FUNCTION_BLOCK FB_TVRModbusMaster
VAR_INPUT
END_VAR
VAR_OUTPUT
END_VAR
VAR
	fbModbusRTUMaster : ModbusRtuMaster_KL6x22B;	//Modbus RTU Master
	
	nUnitID			:	BYTE :=	0;	//Modbus device ID
	
	//Modbus Registers
	nRegSetpoint	:	WORD := 0;
	nRegForce		:	WORD := 1;
	nRegActual		:	WORD := 7;
	
	//Properties
	bError 			: 	BOOL := FALSE;
	fNominalVolFlow	: 	REAL := 3690;
	fVolFlowSet 	: 	REAL := 0;
	fVolFlowAct		: 	REAL;
	
	//Internal vars
	bFlagForce		:	BOOL := FALSE;
	bModErr 		: 	BOOL;
	ErrID 			: 	MODBUS_ERRORS;
	fRelFlowMax		:	WORD := 10000;
	fRelFlowMin		:	WORD := 1024;
	nForce			:	WORD := 0;
	fSetModbus		:	WORD := fRelFlowMin;
	sVolFlowAct		: 	WORD;
	
	//Timer
	Tim			:	TON;
	
	//State
	nState		:	INT	:= 1;
	
END_VAR

PROPERTY Error : Bool
GET
Error := THIS^.bError;
END_GET
SET
THIS^.bError := Error;
END_SET
END_PROPERTY

PROPERTY NominalVolumeFlow : REAL
GET
NominalVolumeFlow := THIS^.fNominalVolFlow;
END_GET
SET
THIS^.fNominalVolFlow := NominalVolumeFlow;
END_SET
END_PROPERTY

METHOD Run : BOOL
VAR_INPUT
END_VAR

VAR
	END_I: INT;
END_VAR
Tim(PT:=T#100MS,IN:=TRUE);
	IF Tim.Q THEN
		Tim(IN:=FALSE);

		CASE nState OF
			//Force or release force
			1: //Initialize writing force or release
				IF NOT fbModbusRTUMaster.BUSY THEN
					//IF setpoint is 0, force close ELSE release force mode
					IF fVolFlowSet = 0 OR bFlagForce = TRUE THEN
						//Force close
						nForce := 2;
						//Initialize writing process
						fbModbusRTUMaster.WriteSingleRegister(	UnitID		:=	nUnitID,				//Modbus ID of device
																MBAddr		:=	nRegForce,				//Register address,
																Quantity	:=	1,						//Number of registers to be written
																pMemoryAddr	:=	ADR(nForce),			//Pointer to write data
																cbLength	:=	SIZEOF(fVolFlowSet),	//Size of write data
																Timeout		:=	T#5S,					//Time to wait for the slave to respond
																Execute		:=	TRUE
															);
					ELSE
						//Release force close
						nForce := 0;
						//Initialize writing process
						fbModbusRTUMaster.WriteSingleRegister(	UnitID		:=	nUnitID,				//Modbus ID of device
																MBAddr		:=	nRegForce,				//Register address,
																Quantity	:=	1,						//Number of registers to be written
																pMemoryAddr	:=	ADR(nForce),			//Pointer to write data
																cbLength	:=	SIZEOF(fVolFlowSet),	//Size of write data
																Timeout		:=	T#5S,					//Time to wait for the slave to respond
																Execute		:=	TRUE
															);
					END_IF
				END_IF
				nState := 2;
				Run := FALSE;
				
			2:	//Finish writing force or release
				fbModbusRTUMaster.WriteSingleRegister(Execute:=FALSE, Error=>bModErr, ErrorID=>ErrID);
				IF NOT fbModbusRTUMaster.BUSY THEN
					nState := 3;
				END_IF
				Run := FALSE;
				
			3:	//Setpoint writing
				IF NOT fbModbusRTUMaster.BUSY THEN
					//Check operational limits
					IF fVolFlowSet < fRelFlowMin/fRelFlowMax*fNominalVolFlow THEN
						fVolFlowSet := fRelFlowMin/fRelFlowMax*fNominalVolFlow; //Set to minimum allowed volume flow
					ELSIF fVolFlowSet > fNominalVolFlow THEN
						fVolFlowSet := fNominalVolFlow; //Set to maximum allowed volumen flow
					ELSE
						//do nothing
					END_IF
					//Write setpoint
					//fSetModbus := REAL_TO_WORD(fRelFlowMax*(fVolFlowSet-(fRelFlowMin/fRelFlowMax*fNominalVolFlow))/(fNominalVolFlow-fRelFlowMin));
					fSetModbus := REAL_TO_WORD(fRelFlowMax*fVolFlowSet/fNominalVolFlow);
					//Initialize writing process
					fbModbusRTUMaster.WriteSingleRegister(	UnitID		:=	nUnitID,				//Modbus ID of device
															MBAddr		:=	nRegSetpoint,			//Register address
															Quantity	:=	1,						//Number of registers to be written
															pMemoryAddr	:=	ADR(fSetModbus),		//Pointer to write data
															cbLength	:=	SIZEOF(fSetModbus),		//Size of write data
															Timeout		:=	T#5S,					//Time to wait for the slave to respond
															Execute		:=	TRUE
														);
				END_IF
				nState := 4;
				Run := FALSE;

			4: //Finish writing	
				fbModbusRTUMaster.WriteSingleRegister(Execute:=FALSE, Error=>bModErr, ErrorID=>ErrID);
				IF NOT fbModbusRTUMaster.BUSY THEN
					nState := 5;
				END_IF
				Run := FALSE;
					
			5: //Start reading
				IF NOT fbModbusRTUMaster.BUSY THEN
					//Initialize reading process
					fbModbusRTUMaster.ReadRegs(	UnitID		:=	nUnitID,				//Modbus ID of device
												MBAddr		:=	nRegActual,				//Register address
												Quantity	:=	1,						//Number of registers to be read
												pMemoryAddr	:=	ADR(sVolFlowAct),		//Pointer to read data
												cbLength	:=	SIZEOF(sVolFlowAct),	//Size of read data
												Timeout		:=	T#5S,					//Time to wait for the slave to respond
												Execute		:=	TRUE
												);
				ELSE
					//do nothing
				END_IF
				nState := 6;
				Run := FALSE;
				
			6: //Finish reading
				fbModbusRTUMaster.ReadRegs(Execute:=FALSE, Error=>bModErr, ErrorID=>ErrID);
				IF NOT fbModbusRTUMaster.BUSY THEN
					fVolFlowAct := WORD_TO_REAL(sVolFlowAct);
					nState := 1;
					Run := TRUE;
				ELSE
					Run := FALSE;
				END_IF
				
		END_CASE
		
END_IF
END_METHOD

PROPERTY UnitID : BYTE
GET
UnitID := THIS^.nUnitID;
END_GET
SET
THIS^.nUnitID := UnitID;
END_SET
END_PROPERTY

PROPERTY VolumeFlowActual : REAL
GET
VolumeFlowActual := THIS^.fVolFlowAct;
END_GET
SET
THIS^.fVolFlowAct := VolumeFlowActual;
END_SET
END_PROPERTY

PROPERTY VolumeFlowSetpoint : REAL
GET
VolumeFlowSetpoint := THIS^.fVolFlowSet;
END_GET
SET
THIS^.fVolFlowSet := VolumeFlowSetpoint;
END_SET
END_PROPERTY

END_FUNCTION_BLOCK

(* stored: Version 1.1.0.1, ProductVersion 3.1.4024.0
   POU FB_TVRModbusMaster: Id {60646394-1a33-45bb-968b-5091f0cf2467}, SpecialFunc None
   Property Error: Id {2712f295-a784-4b32-a7f9-34003f757e09}
   Get Get: Id {1246bcd0-d7de-4218-b62b-b1d303a5361e}
   Set Set: Id {e41e6059-501e-4279-9af4-2c7583f67d73}
   Property NominalVolumeFlow: Id {5f693b9b-b75b-4809-a86d-4c62834407cb}
   Get Get: Id {05ff600d-aa92-4406-bda2-cedabeba8351}
   Set Set: Id {1dc5ca52-92f9-46ee-bcb7-937e09f178ac}
   Method Run: Id {ac2cb6c2-a0db-485f-bb8a-acbeb92cc7df}
   Property UnitID: Id {9f8b936f-964a-4ae4-97fc-cfb51b36d120}
   Get Get: Id {796bd35f-f665-4674-8990-f75f70a4592b}
   Set Set: Id {521d08d8-dd9f-4a87-995f-31a8deea0ad4}
   Property VolumeFlowActual: Id {29020dfb-61ba-491f-a514-72868efd643c}
   Get Get: Id {49e52031-720c-4dd1-b948-2548533c359e}
   Set Set: Id {506a82c6-5c0c-4090-b0bd-9f1d2674b877}
   Property VolumeFlowSetpoint: Id {819b1658-a701-40d9-9baa-1e13e90a04e3}
   Get Get: Id {f7df6e47-76d8-429c-a22b-4dcb0e8a27f5}
   Set Set: Id {1c8abb76-b064-40ef-ac2c-f28ad267b127} *)
